DATA_BLOCK "DB_Z220_3_HMI"
{ DB_Accessible_From_OPC_UA := 'FALSE' ;
 DB_Accessible_From_Webserver := 'FALSE' ;
 S7_Optimized_Access := 'FALSE' }
VERSION : 0.1
NON_RETAIN
   STRUCT
      tAlm : Struct   // HMI Alarms
         tE : Struct   // Emergency alarms
            xSpare_0 : Bool;
            xSpare_1 : Bool;
            xSpare_2 : Bool;
            xSpare_3 : Bool;
            xSpare_4 : Bool;
            xSpare_5 : Bool;
            xSpare_6 : Bool;
            xSpare_7 : Bool;
            xSpare_8 : Bool;
            xSpare_9 : Bool;
            xSpare_10 : Bool;
            xSpare_11 : Bool;
            xSpare_12 : Bool;
            xSpare_13 : Bool;
            xSpare_14 : Bool;
            xSpare_15 : Bool;
            xSpare_16 : Bool;
            xSpare_17 : Bool;
            xSpare_18 : Bool;
            xSpare_19 : Bool;
            xSpare_20 : Bool;
            xSpare_21 : Bool;
            xSpare_22 : Bool;
            xSpare_23 : Bool;
            xSpare_24 : Bool;
            xSpare_25 : Bool;
            xSpare_26 { ExternalAccessible := 'False'; ExternalVisible := 'False'; ExternalWritable := 'False'} : Bool;
            xSpare_27 { ExternalAccessible := 'False'; ExternalVisible := 'False'; ExternalWritable := 'False'} : Bool;
            xSpare_28 { ExternalAccessible := 'False'; ExternalVisible := 'False'; ExternalWritable := 'False'} : Bool;
            xSpare_29 { ExternalAccessible := 'False'; ExternalVisible := 'False'; ExternalWritable := 'False'} : Bool;
            xSpare_30 { ExternalAccessible := 'False'; ExternalVisible := 'False'; ExternalWritable := 'False'} : Bool;
            xSpare_31 { ExternalAccessible := 'False'; ExternalVisible := 'False'; ExternalWritable := 'False'} : Bool;
         END_STRUCT;
         tS : Struct   // Stopping faults
            xSpare_0 : Bool;   //
            xSpare_1 : Bool;
            xSpare_2 : Bool;
            xSpare_3 : Bool;
            xSpare_4 : Bool;
            xSpare_5 : Bool;
            xSpare_6 : Bool;
            xSpare_7 : Bool;
            xSpare_8 : Bool;
            xSpare_9 : Bool;
            xSpare_10 : Bool;
            xSpare_11 : Bool;
            xSpare_12 : Bool;
            xSpare_13 : Bool;
            xSpare_14 : Bool;
            xSpare_15 : Bool;
            xSpare_16 : Bool;
            xSpare_17 : Bool;
            xSpare_18 : Bool;
            xSpare_19 : Bool;
            xSpare_20 : Bool;
            xSpare_21 : Bool;
            xSpare_22 : Bool;
            xSpare_23 : Bool;
            xSpare_24 : Bool;
            xSpare_25 : Bool;
            xSpare_26 : Bool;
            xSpare_27 : Bool;
            xSpare_28 : Bool;
            xSpare_29 : Bool;
            xSpare_30 : Bool;
            xSpare_31 : Bool;
         END_STRUCT;
         tF : Struct   // Faults
            x0 : Bool;   // B.Check spray ink carriage
            x2 : Bool;   // SL.Ink tank empty
            x1 : Bool;   // B.Check spray ink carriage dirty lens
            xSpare_3 : Bool;
            xSpare_4 : Bool;
            xSpare_5 : Bool;
            xSpare_6 : Bool;
            xSpare_7 : Bool;
            xSpare_8 : Bool;
            xSpare_9 : Bool;
            xSpare_10 : Bool;
            xSpare_11 : Bool;
            xSpare_12 : Bool;
            xSpare_13 : Bool;
            xSpare_14 : Bool;
            xSpare_15 : Bool;
            xSpare_16 : Bool;
            xSpare_17 : Bool;   //
            xSpare_18 : Bool;
            xSpare_19 : Bool;
            xSpare_20 : Bool;
            xSpare_21 : Bool;
            xSpare_22 : Bool;
            xSpare_23 : Bool;
            xSpare_24 : Bool;
            xSpare_25 : Bool;
            xSpare_26 : Bool;
            xSpare_27 : Bool;
            xSpare_28 : Bool;
            xSpare_29 : Bool;
            xSpare_30 : Bool;
            xSpare_31 : Bool;
         END_STRUCT;
         tW : Struct   // Warnings
            xSpare_0 : Bool;
            xSpare_1 : Bool;
            xSpare_2 : Bool;
            xSpare_3 : Bool;
            xSpare_4 : Bool;
            xSpare_5 : Bool;
            xSpare_6 : Bool;
            xSpare_7 : Bool;
            xSpare_8 : Bool;
            xSpare_9 : Bool;
            xSpare_10 : Bool;
            xSpare_11 : Bool;
            xSpare_12 : Bool;
            xSpare_13 : Bool;
            xSpare_14 : Bool;
            xSpare_15 : Bool;
            xSpare_16 : Bool;
            xSpare_17 : Bool;
            xSpare_18 : Bool;
            xSpare_19 : Bool;
            xSpare_20 : Bool;
            xSpare_21 : Bool;
            xSpare_22 : Bool;
            xSpare_23 : Bool;
            xSpare_24 : Bool;
            xSpare_25 : Bool;
            xSpare_26 : Bool;
            xSpare_27 : Bool;
            xSpare_28 : Bool;
            xSpare_29 : Bool;
            xSpare_30 : Bool;
            xSpare_31 : Bool;
         END_STRUCT;
      END_STRUCT;
      tHMR { ExternalWritable := 'False'} : Struct   // HMI Read
         xSpare0 { ExternalWritable := 'False'} : Bool;
         xSpare1 { ExternalWritable := 'False'} : Bool;
         xSpare2 { ExternalWritable := 'False'} : Bool;
         xSpare3 { ExternalWritable := 'False'} : Bool;
         xSpare4 { ExternalWritable := 'False'} : Bool;
         xSpare5 { ExternalWritable := 'False'} : Bool;
         xSpare6 { ExternalWritable := 'False'} : Bool;
         xSpare7 { ExternalWritable := 'False'} : Bool;
         xSpare8 { ExternalWritable := 'False'} : Bool;
         xSpare9 { ExternalWritable := 'False'} : Bool;
         xSpare10 { ExternalWritable := 'False'} : Bool;
         xSpare11 { ExternalWritable := 'False'} : Bool;
         xSpare12 { ExternalWritable := 'False'} : Bool;
         xSpare13 { ExternalWritable := 'False'} : Bool;
         xSpare14 { ExternalWritable := 'False'} : Bool;
         xSpare15 { ExternalWritable := 'False'} : Bool;   //
         xSpare16 { ExternalWritable := 'False'} : Bool;
         xSpare17 { ExternalWritable := 'False'} : Bool;
         xSpare18 { ExternalWritable := 'False'} : Bool;
         xSpare19 { ExternalWritable := 'False'} : Bool;
         xSpare20 { ExternalWritable := 'False'} : Bool;
         xSpare21 { ExternalWritable := 'False'} : Bool;
         xSpare22 { ExternalWritable := 'False'} : Bool;
         xSpare23 { ExternalWritable := 'False'} : Bool;
         xSpare24 { ExternalWritable := 'False'} : Bool;
         xSpare25 { ExternalWritable := 'False'} : Bool;
         xSpare26 { ExternalWritable := 'False'} : Bool;
         xSpare27 { ExternalWritable := 'False'} : Bool;
         xSpare28 { ExternalWritable := 'False'} : Bool;
         xSpare29 { ExternalWritable := 'False'} : Bool;
         xSpare30 { ExternalWritable := 'False'} : Bool;
         xSpare31 { ExternalWritable := 'False'} : Bool;
         xSpare { ExternalWritable := 'False'} : Array[0..15] of Bool;
         iSpare0 { ExternalWritable := 'False'} : Int;
         iSpare1 { ExternalWritable := 'False'} : Int;
         iSpare2 { ExternalWritable := 'False'} : Int;
         iSpare3 { ExternalWritable := 'False'} : Int;
         iSpare4 { ExternalWritable := 'False'} : Int;
         iSpare5 { ExternalWritable := 'False'} : Int;
         iSpare6 { ExternalWritable := 'False'} : Int;
         iSpare7 { ExternalWritable := 'False'} : Int;
         iSpare8 { ExternalWritable := 'False'} : Int;
         iSpare9 { ExternalWritable := 'False'} : Int;
         iSpare10 { ExternalWritable := 'False'} : Int;
         iSpare11 { ExternalWritable := 'False'} : Int;
         iSpare12 { ExternalWritable := 'False'} : Int;
         iSpare13 { ExternalWritable := 'False'} : Int;
         iSpare14 { ExternalWritable := 'False'} : Int;
         iSpare15 { ExternalWritable := 'False'} : Int;
         iSpare16 { ExternalWritable := 'False'} : Int;
         dZoneMode { ExternalWritable := 'False'} : DInt;   // Zone modality (1=Manual;4=Automatic;8=Manual request) {x|x|x|x|O}
         dProdModeRequest { ExternalWritable := 'False'} : DInt;   // Production modality request (1=Out of Production 3= In production) {x|x|x|x|O}
         dProdModeActual { ExternalWritable := 'False'} : DInt;   // Production modality actual (1=Out of production 3=In production 8=Out of production request 9=In production request) {x|x|x|x|O}
         dActualDistanceFromSnaproll { ExternalWritable := 'False'} : DInt;   // Actual distance from snaproll [mm/100] {x|x|x|x|O}
         dSprayCounter { ExternalWritable := 'False'} : DInt;
         dPhSprayCounter { ExternalWritable := 'False'} : DInt;
         dEvReactionTime { ExternalWritable := 'False'} : DInt;
         dCalibDeltaXPosition_cmm { ExternalWritable := 'False'} : DInt;   // Calibration.Theorical spray position X [mm/100] {mm/100|mm|0|7000|M}
         dCalibDeltaYPosition_cmm { ExternalWritable := 'False'} : DInt;   // Calibration.Theorical spray position Y [mm/100] {mm/100|mm|0|7000|M}
         dSpare9 { ExternalWritable := 'False'} : DInt;
         dSpare10 { ExternalWritable := 'False'} : DInt;
         dSpare11 { ExternalWritable := 'False'} : DInt;
         dSpare12 { ExternalWritable := 'False'} : DInt;
         dSpare13 { ExternalWritable := 'False'} : DInt;
         dSpare14 { ExternalWritable := 'False'} : DInt;
         dSpare15 { ExternalWritable := 'False'} : DInt;
         rSpare0 { ExternalWritable := 'False'} : Real;
         rSpare1 { ExternalWritable := 'False'} : Real;
         rSpare2 { ExternalWritable := 'False'} : Real;
         rSpare3 { ExternalWritable := 'False'} : Real;
         rSpare4 { ExternalWritable := 'False'} : Real;
         rSpare5 { ExternalWritable := 'False'} : Real;
         rSpare6 { ExternalWritable := 'False'} : Real;
         rSpare7 { ExternalWritable := 'False'} : Real;
         rSpare8 { ExternalWritable := 'False'} : Real;
         tManCmd { ExternalWritable := 'False'} : Struct
            xSpare0 { ExternalWritable := 'False'} : Bool;   //
            xSpare1 { ExternalWritable := 'False'} : Bool;
            xSpare2 { ExternalWritable := 'False'} : Bool;
            xSpare3 { ExternalWritable := 'False'} : Bool;
            xSpare4 { ExternalWritable := 'False'} : Bool;
            xSpare5 { ExternalWritable := 'False'} : Bool;
            xSpare6 { ExternalWritable := 'False'} : Bool;
            xSpare7 { ExternalWritable := 'False'} : Bool;
            xSpare8 { ExternalWritable := 'False'} : Bool;
            xSpare9 { ExternalWritable := 'False'} : Bool;
            xSpare10 { ExternalWritable := 'False'} : Bool;
            xSpare11 { ExternalWritable := 'False'} : Bool;
            xSpare12 { ExternalWritable := 'False'} : Bool;
            xSpare13 { ExternalWritable := 'False'} : Bool;
            xSpare14 { ExternalWritable := 'False'} : Bool;
            xSpare15 { ExternalWritable := 'False'} : Bool;
            xSpare { ExternalWritable := 'False'} : Array[0..15] of Bool;
         END_STRUCT;
      END_STRUCT;
      tHMW : Struct   // HMI Write
         xAutoModeReq : Bool;   // Automatic mode request {x|x|x|x|O}
         xManModeReq : Bool;   // Manual mode request {x|x|x|x|O}
         xUpdateDistanceFromSnapRoll : Bool;   // Update Distance From Snap Roll {x|x|x|x|M}
         xCalibrate : Bool;   // Calibrate spray position {x|x|x|x|M}
         xCleaningCycle : Bool;   // Cleaning cycle enabled {x|x|x|x|O}
         xSprayOnBreakEnabled : Bool;   // Spray during glass break {x|x|x|x|O}
         xSprayCheckEnabled : Bool;   // Spray check enabled {x|x|x|x|O}
         xResetCounter : Bool;
         xSpare8 : Bool;
         xSpare9 { ExternalWritable := 'False'} : Bool;
         xSpare10 : Bool;
         xSpare11 : Bool;
         xSpare12 : Bool;
         xSpare13 : Bool;
         xSpare14 : Bool;
         xSpare15 : Bool;   //
         xSpare16 : Bool;   //
         xSpare17 : Bool;
         xSpare18 : Bool;
         xSpare19 : Bool;
         xSpare20 : Bool;
         xSpare21 : Bool;
         xSpare22 : Bool;
         xSpare23 : Bool;
         xSpare24 : Bool;
         xSpare25 : Bool;
         xSpare26 : Bool;
         xSpare27 : Bool;
         xSpare28 : Bool;
         xSpare29 : Bool;
         xSpare30 : Bool;
         xSpare31 : Bool;
         xSpare : Array[0..15] of Bool;
         iSpare0 : Int;
         iSpare1 : Int;
         iSpare2 : Int;
         iSpare3 : Int;
         iSpare4 : Int;
         iSpare5 : Int;
         iSpare6 : Int;
         iSpare7 : Int;
         iSpare8 : Int;
         iSpare9 : Int;
         iSpare10 : Int;
         iSpare11 : Int;
         iSpare12 : Int;
         iSpare13 : Int;
         iSpare14 : Int;
         iSpare15 : Int;
         iSpare16 : Int;
         dDistanceFromSnaproll_cmm : DInt;   // Distance from snaproll [mm/100] {x|x|x|x|O}
         dSpare1 : DInt;   //
         dCleaningInterval_ms : DInt;   // Cleaning cycle interval [ms] {ms|s|3600|36000|O}
         dSpraySpace_cmm : DInt;   // Spray space [mm/100] {mm/100|mm|1|100|O}
         dSprayReactionTimeON_ms : DInt;   // Spray reaction time [ms] {ms|s|0.001|2|M}
         dSprayReactionTimeOFF_ms : DInt;   // Spray reaction time off [ms] {ms|s|0.001|2|M}
         dCalibDefectMeasXPosition_cmm : DInt;   // Calibration.Measured defect position X [mm/100] {mm/100|mm|0|7000|M}
         dCalibSprayMeasXPosition_cmm : DInt;   // Calibration.Measured spray position X [mm/100] {mm/100|mm|0|7000|M}
         dCalibDefectMeasYPosition_cmm : DInt;   // Calibration.Measured defect position Y [mm/100] {mm/100|mm|0|7000|M}
         dCalibSprayMeasYPosition_cmm : DInt;   // Calibration.Measured spray position Y [mm/100] {mm/100|mm|0|7000|M}
         dSpare10 : DInt;
         dSpare11 : DInt;
         dSpare12 : DInt;
         dSpare13 : DInt;
         dSpare14 : DInt;
         dSpare15 : DInt;
         dSpare16 : DInt;
         rSpare0 : Real;
         rSpare1 : Real;
         rSpare2 : Real;
         rSpare3 : Real;
         rSpare4 : Real;
         rSpare5 : Real;
         rSpare6 : Real;
         rSpare7 : Real;
         rSpare8 : Real;
         tManCmd : Struct
            xSpare0 : Bool;
            xSpare1 : Bool;
            xSpare2 { ExternalWritable := 'False'} : Bool;
            xSpare3 { ExternalWritable := 'False'} : Bool;
            xSpare4 { ExternalWritable := 'False'} : Bool;
            xSpare5 { ExternalWritable := 'False'} : Bool;
            xSpare6 { ExternalWritable := 'False'} : Bool;
            xSpare7 { ExternalWritable := 'False'} : Bool;
            xSpare8 { ExternalWritable := 'False'} : Bool;
            xSpare9 { ExternalWritable := 'False'} : Bool;
            xSpare10 { ExternalWritable := 'False'} : Bool;
            xSpare11 { ExternalWritable := 'False'} : Bool;
            xSpare12 { ExternalWritable := 'False'} : Bool;
            xSpare13 { ExternalWritable := 'False'} : Bool;
            xSpare14 { ExternalWritable := 'False'} : Bool;
            xSpare15 { ExternalWritable := 'False'} : Bool;
            xSpare16 : Bool;
            xSpare17 : Bool;
            xSpare18 : Bool;
            xSpare19 : Bool;
            xSpare20 : Bool;
            xSpare21 : Bool;
            xSpare22 : Bool;
            xSpare23 : Bool;
            xSpare24 : Bool;
            xSpare25 : Bool;
            xSpare26 : Bool;
            xSpare27 : Bool;
            xSpare28 : Bool;
            xSpare29 : Bool;
            xSpare30 : Bool;
            xSpare31 : Bool;
         END_STRUCT;
      END_STRUCT;
   END_STRUCT;


BEGIN
   tAlm.tE.xSpare_0 := TRUE;
   tAlm.tE.xSpare_1 := TRUE;
   tAlm.tE.xSpare_2 := TRUE;
   tAlm.tE.xSpare_3 := TRUE;
   tAlm.tE.xSpare_4 := TRUE;
   tAlm.tE.xSpare_5 := TRUE;
   tAlm.tE.xSpare_6 := TRUE;
   tAlm.tE.xSpare_7 := TRUE;
   tAlm.tE.xSpare_8 := TRUE;
   tAlm.tE.xSpare_9 := TRUE;
   tAlm.tE.xSpare_10 := FALSE;
   tAlm.tE.xSpare_11 := FALSE;
   tAlm.tE.xSpare_12 := FALSE;
   tAlm.tE.xSpare_13 := FALSE;
   tAlm.tE.xSpare_14 := FALSE;
   tAlm.tE.xSpare_15 := FALSE;
   tAlm.tE.xSpare_16 := FALSE;
   tAlm.tE.xSpare_17 := FALSE;
   tAlm.tE.xSpare_18 := FALSE;
   tAlm.tE.xSpare_19 := FALSE;
   tAlm.tE.xSpare_20 := FALSE;
   tAlm.tE.xSpare_21 := FALSE;
   tAlm.tE.xSpare_22 := FALSE;
   tAlm.tE.xSpare_23 := FALSE;
   tAlm.tE.xSpare_24 := FALSE;
   tAlm.tE.xSpare_25 := FALSE;
   tAlm.tE.xSpare_26 := FALSE;
   tAlm.tE.xSpare_27 := FALSE;
   tAlm.tE.xSpare_28 := FALSE;
   tAlm.tE.xSpare_29 := FALSE;
   tAlm.tE.xSpare_30 := FALSE;
   tAlm.tE.xSpare_31 := FALSE;
   tAlm.tS.xSpare_0 := FALSE;
   tAlm.tS.xSpare_1 := FALSE;
   tAlm.tS.xSpare_2 := FALSE;
   tAlm.tS.xSpare_3 := FALSE;
   tAlm.tS.xSpare_4 := FALSE;
   tAlm.tS.xSpare_5 := FALSE;
   tAlm.tS.xSpare_6 := FALSE;
   tAlm.tS.xSpare_7 := FALSE;
   tAlm.tS.xSpare_8 := FALSE;
   tAlm.tS.xSpare_9 := FALSE;
   tAlm.tS.xSpare_10 := FALSE;
   tAlm.tS.xSpare_11 := FALSE;
   tAlm.tS.xSpare_12 := FALSE;
   tAlm.tS.xSpare_13 := FALSE;
   tAlm.tS.xSpare_14 := FALSE;
   tAlm.tS.xSpare_15 := FALSE;
   tAlm.tS.xSpare_16 := FALSE;
   tAlm.tS.xSpare_17 := FALSE;
   tAlm.tS.xSpare_18 := FALSE;
   tAlm.tS.xSpare_19 := FALSE;
   tAlm.tS.xSpare_20 := FALSE;
   tAlm.tS.xSpare_21 := FALSE;
   tAlm.tS.xSpare_22 := FALSE;
   tAlm.tS.xSpare_23 := FALSE;
   tAlm.tS.xSpare_24 := FALSE;
   tAlm.tS.xSpare_25 := FALSE;
   tAlm.tS.xSpare_26 := FALSE;
   tAlm.tS.xSpare_27 := FALSE;
   tAlm.tS.xSpare_28 := FALSE;
   tAlm.tS.xSpare_29 := FALSE;
   tAlm.tS.xSpare_30 := FALSE;
   tAlm.tS.xSpare_31 := FALSE;
   tAlm.tF.xSpare_3 := FALSE;
   tAlm.tF.xSpare_4 := FALSE;
   tAlm.tF.xSpare_5 := FALSE;
   tAlm.tF.xSpare_6 := FALSE;
   tAlm.tF.xSpare_7 := FALSE;
   tAlm.tF.xSpare_8 := FALSE;
   tAlm.tF.xSpare_9 := FALSE;
   tAlm.tF.xSpare_10 := FALSE;
   tAlm.tF.xSpare_11 := FALSE;
   tAlm.tF.xSpare_20 := FALSE;
   tAlm.tF.xSpare_21 := FALSE;
   tAlm.tF.xSpare_22 := FALSE;
   tAlm.tF.xSpare_23 := FALSE;
   tAlm.tF.xSpare_24 := FALSE;
   tAlm.tF.xSpare_25 := FALSE;
   tAlm.tF.xSpare_26 := FALSE;
   tAlm.tF.xSpare_27 := FALSE;
   tAlm.tF.xSpare_28 := FALSE;
   tAlm.tF.xSpare_29 := FALSE;
   tAlm.tF.xSpare_30 := FALSE;
   tAlm.tF.xSpare_31 := FALSE;
   tAlm.tW.xSpare_0 := FALSE;
   tAlm.tW.xSpare_1 := FALSE;
   tAlm.tW.xSpare_2 := FALSE;
   tAlm.tW.xSpare_3 := FALSE;
   tAlm.tW.xSpare_4 := FALSE;
   tAlm.tW.xSpare_5 := FALSE;
   tAlm.tW.xSpare_6 := FALSE;
   tAlm.tW.xSpare_7 := FALSE;
   tAlm.tW.xSpare_8 := FALSE;
   tAlm.tW.xSpare_9 := FALSE;
   tAlm.tW.xSpare_10 := FALSE;
   tAlm.tW.xSpare_11 := FALSE;
   tAlm.tW.xSpare_12 := FALSE;
   tAlm.tW.xSpare_13 := FALSE;
   tAlm.tW.xSpare_14 := FALSE;
   tAlm.tW.xSpare_15 := FALSE;
   tAlm.tW.xSpare_16 := FALSE;
   tAlm.tW.xSpare_17 := FALSE;
   tAlm.tW.xSpare_18 := FALSE;
   tAlm.tW.xSpare_19 := FALSE;
   tAlm.tW.xSpare_20 := FALSE;
   tAlm.tW.xSpare_21 := FALSE;
   tAlm.tW.xSpare_22 := FALSE;
   tAlm.tW.xSpare_23 := FALSE;
   tAlm.tW.xSpare_24 := FALSE;
   tAlm.tW.xSpare_25 := FALSE;
   tAlm.tW.xSpare_26 := FALSE;
   tAlm.tW.xSpare_27 := FALSE;
   tAlm.tW.xSpare_28 := FALSE;
   tAlm.tW.xSpare_29 := FALSE;
   tAlm.tW.xSpare_30 := FALSE;
   tAlm.tW.xSpare_31 := FALSE;
   tHMR.xSpare15 := FALSE;
   tHMW.xSpare15 := FALSE;
   tHMW.xSpare16 := FALSE;

END_DATA_BLOCK

DATA_BLOCK "DB_Z220_2_HMI"
{ DB_Accessible_From_OPC_UA := 'FALSE' ;
 DB_Accessible_From_Webserver := 'FALSE' ;
 S7_Optimized_Access := 'FALSE' }
VERSION : 0.1
NON_RETAIN
   STRUCT
      tAlm : Struct   // HMI Alarms
         tE : Struct   // Emergency alarms
            xSpare_0 : Bool;
            xSpare_1 : Bool;
            xSpare_2 : Bool;
            xSpare_3 : Bool;
            xSpare_4 : Bool;
            xSpare_5 : Bool;
            xSpare_6 : Bool;
            xSpare_7 : Bool;
            xSpare_8 : Bool;
            xSpare_9 : Bool;
            xSpare_10 : Bool;
            xSpare_11 : Bool;
            xSpare_12 : Bool;
            xSpare_13 : Bool;
            xSpare_14 : Bool;
            xSpare_15 : Bool;
            xSpare_16 : Bool;
            xSpare_17 : Bool;
            xSpare_18 : Bool;
            xSpare_19 : Bool;
            xSpare_20 : Bool;
            xSpare_21 : Bool;
            xSpare_22 : Bool;
            xSpare_23 : Bool;
            xSpare_24 : Bool;
            xSpare_25 : Bool;
            xSpare_26 { ExternalAccessible := 'False'; ExternalVisible := 'False'; ExternalWritable := 'False'} : Bool;
            xSpare_27 { ExternalAccessible := 'False'; ExternalVisible := 'False'; ExternalWritable := 'False'} : Bool;
            xSpare_28 { ExternalAccessible := 'False'; ExternalVisible := 'False'; ExternalWritable := 'False'} : Bool;
            xSpare_29 { ExternalAccessible := 'False'; ExternalVisible := 'False'; ExternalWritable := 'False'} : Bool;
            xSpare_30 { ExternalAccessible := 'False'; ExternalVisible := 'False'; ExternalWritable := 'False'} : Bool;
            xSpare_31 { ExternalAccessible := 'False'; ExternalVisible := 'False'; ExternalWritable := 'False'} : Bool;
         END_STRUCT;
         tS : Struct   // Stopping faults
            xSpare_0 : Bool;   //
            xSpare_1 : Bool;
            xSpare_2 : Bool;
            xSpare_3 : Bool;
            xSpare_4 : Bool;
            xSpare_5 : Bool;
            xSpare_6 : Bool;
            xSpare_7 : Bool;
            xSpare_8 : Bool;
            xSpare_9 : Bool;
            xSpare_10 : Bool;
            xSpare_11 : Bool;
            xSpare_12 : Bool;
            xSpare_13 : Bool;
            xSpare_14 : Bool;
            xSpare_15 : Bool;
            xSpare_16 : Bool;
            xSpare_17 : Bool;
            xSpare_18 : Bool;
            xSpare_19 : Bool;
            xSpare_20 : Bool;
            xSpare_21 : Bool;
            xSpare_22 : Bool;
            xSpare_23 : Bool;
            xSpare_24 : Bool;
            xSpare_25 : Bool;
            xSpare_26 : Bool;
            xSpare_27 : Bool;
            xSpare_28 : Bool;
            xSpare_29 : Bool;
            xSpare_30 : Bool;
            xSpare_31 : Bool;
         END_STRUCT;
         tF : Struct   // Faults
            x0 : Bool;   // B.Check spray ink carriage
            x2 : Bool;   // SL.Ink tank empty
            x1 : Bool;   // B.Check spray ink carriage dirty lens
            xSpare_3 : Bool;
            xSpare_4 : Bool;
            xSpare_5 : Bool;
            xSpare_6 : Bool;
            xSpare_7 : Bool;
            xSpare_8 : Bool;
            xSpare_9 : Bool;
            xSpare_10 : Bool;
            xSpare_11 : Bool;
            xSpare_12 : Bool;
            xSpare_13 : Bool;
            xSpare_14 : Bool;
            xSpare_15 : Bool;
            xSpare_16 : Bool;
            xSpare_17 : Bool;   //
            xSpare_18 : Bool;
            xSpare_19 : Bool;
            xSpare_20 : Bool;
            xSpare_21 : Bool;
            xSpare_22 : Bool;
            xSpare_23 : Bool;
            xSpare_24 : Bool;
            xSpare_25 : Bool;
            xSpare_26 : Bool;
            xSpare_27 : Bool;
            xSpare_28 : Bool;
            xSpare_29 : Bool;
            xSpare_30 : Bool;
            xSpare_31 : Bool;
         END_STRUCT;
         tW : Struct   // Warnings
            xSpare_0 : Bool;
            xSpare_1 : Bool;
            xSpare_2 : Bool;
            xSpare_3 : Bool;
            xSpare_4 : Bool;
            xSpare_5 : Bool;
            xSpare_6 : Bool;
            xSpare_7 : Bool;
            xSpare_8 : Bool;
            xSpare_9 : Bool;
            xSpare_10 : Bool;
            xSpare_11 : Bool;
            xSpare_12 : Bool;
            xSpare_13 : Bool;
            xSpare_14 : Bool;
            xSpare_15 : Bool;
            xSpare_16 : Bool;
            xSpare_17 : Bool;
            xSpare_18 : Bool;
            xSpare_19 : Bool;
            xSpare_20 : Bool;
            xSpare_21 : Bool;
            xSpare_22 : Bool;
            xSpare_23 : Bool;
            xSpare_24 : Bool;
            xSpare_25 : Bool;
            xSpare_26 : Bool;
            xSpare_27 : Bool;
            xSpare_28 : Bool;
            xSpare_29 : Bool;
            xSpare_30 : Bool;
            xSpare_31 : Bool;
         END_STRUCT;
      END_STRUCT;
      tHMR { ExternalWritable := 'False'} : Struct   // HMI Read
         xSpare0 { ExternalWritable := 'False'} : Bool;
         xSpare1 { ExternalWritable := 'False'} : Bool;
         xSpare2 { ExternalWritable := 'False'} : Bool;
         xSpare3 { ExternalWritable := 'False'} : Bool;
         xSpare4 { ExternalWritable := 'False'} : Bool;
         xSpare5 { ExternalWritable := 'False'} : Bool;
         xSpare6 { ExternalWritable := 'False'} : Bool;
         xSpare7 { ExternalWritable := 'False'} : Bool;
         xSpare8 { ExternalWritable := 'False'} : Bool;
         xSpare9 { ExternalWritable := 'False'} : Bool;
         xSpare10 { ExternalWritable := 'False'} : Bool;
         xSpare11 { ExternalWritable := 'False'} : Bool;
         xSpare12 { ExternalWritable := 'False'} : Bool;
         xSpare13 { ExternalWritable := 'False'} : Bool;
         xSpare14 { ExternalWritable := 'False'} : Bool;
         xSpare15 { ExternalWritable := 'False'} : Bool;   //
         xSpare16 { ExternalWritable := 'False'} : Bool;
         xSpare17 { ExternalWritable := 'False'} : Bool;
         xSpare18 { ExternalWritable := 'False'} : Bool;
         xSpare19 { ExternalWritable := 'False'} : Bool;
         xSpare20 { ExternalWritable := 'False'} : Bool;
         xSpare21 { ExternalWritable := 'False'} : Bool;
         xSpare22 { ExternalWritable := 'False'} : Bool;
         xSpare23 { ExternalWritable := 'False'} : Bool;
         xSpare24 { ExternalWritable := 'False'} : Bool;
         xSpare25 { ExternalWritable := 'False'} : Bool;
         xSpare26 { ExternalWritable := 'False'} : Bool;
         xSpare27 { ExternalWritable := 'False'} : Bool;
         xSpare28 { ExternalWritable := 'False'} : Bool;
         xSpare29 { ExternalWritable := 'False'} : Bool;
         xSpare30 { ExternalWritable := 'False'} : Bool;
         xSpare31 { ExternalWritable := 'False'} : Bool;
         xSpare { ExternalWritable := 'False'} : Array[0..15] of Bool;
         iSpare0 { ExternalWritable := 'False'} : Int;
         iSpare1 { ExternalWritable := 'False'} : Int;
         iSpare2 { ExternalWritable := 'False'} : Int;
         iSpare3 { ExternalWritable := 'False'} : Int;
         iSpare4 { ExternalWritable := 'False'} : Int;
         iSpare5 { ExternalWritable := 'False'} : Int;
         iSpare6 { ExternalWritable := 'False'} : Int;
         iSpare7 { ExternalWritable := 'False'} : Int;
         iSpare8 { ExternalWritable := 'False'} : Int;
         iSpare9 { ExternalWritable := 'False'} : Int;
         iSpare10 { ExternalWritable := 'False'} : Int;
         iSpare11 { ExternalWritable := 'False'} : Int;
         iSpare12 { ExternalWritable := 'False'} : Int;
         iSpare13 { ExternalWritable := 'False'} : Int;
         iSpare14 { ExternalWritable := 'False'} : Int;
         iSpare15 { ExternalWritable := 'False'} : Int;
         iSpare16 { ExternalWritable := 'False'} : Int;
         dZoneMode { ExternalWritable := 'False'} : DInt;   // Zone modality (1=Manual;4=Automatic;8=Manual request) {x|x|x|x|O}
         dProdModeRequest { ExternalWritable := 'False'} : DInt;   // Production modality request (1=Out of Production 3= In production) {x|x|x|x|O}
         dProdModeActual { ExternalWritable := 'False'} : DInt;   // Production modality actual (1=Out of production 3=In production 8=Out of production request 9=In production request) {x|x|x|x|O}
         dActualDistanceFromSnaproll { ExternalWritable := 'False'} : DInt;   // Actual distance from snaproll [mm/100] {x|x|x|x|O}
         dSprayCounter { ExternalWritable := 'False'} : DInt;
         dPhSprayCounter { ExternalWritable := 'False'} : DInt;
         dEvReactionTime { ExternalWritable := 'False'} : DInt;
         dCalibDeltaXPosition_cmm { ExternalWritable := 'False'} : DInt;   // Calibration.Theorical spray position X [mm/100] {mm/100|mm|0|7000|M}
         dCalibDeltaYPosition_cmm { ExternalWritable := 'False'} : DInt;   // Calibration.Theorical spray position Y [mm/100] {mm/100|mm|0|7000|M}
         dSpare9 { ExternalWritable := 'False'} : DInt;
         dSpare10 { ExternalWritable := 'False'} : DInt;
         dSpare11 { ExternalWritable := 'False'} : DInt;
         dSpare12 { ExternalWritable := 'False'} : DInt;
         dSpare13 { ExternalWritable := 'False'} : DInt;
         dSpare14 { ExternalWritable := 'False'} : DInt;
         dSpare15 { ExternalWritable := 'False'} : DInt;
         rSpare0 { ExternalWritable := 'False'} : Real;
         rSpare1 { ExternalWritable := 'False'} : Real;
         rSpare2 { ExternalWritable := 'False'} : Real;
         rSpare3 { ExternalWritable := 'False'} : Real;
         rSpare4 { ExternalWritable := 'False'} : Real;
         rSpare5 { ExternalWritable := 'False'} : Real;
         rSpare6 { ExternalWritable := 'False'} : Real;
         rSpare7 { ExternalWritable := 'False'} : Real;
         rSpare8 { ExternalWritable := 'False'} : Real;
         tManCmd { ExternalWritable := 'False'} : Struct
            xSpare0 { ExternalWritable := 'False'} : Bool;   //
            xSpare1 { ExternalWritable := 'False'} : Bool;
            xSpare2 { ExternalWritable := 'False'} : Bool;
            xSpare3 { ExternalWritable := 'False'} : Bool;
            xSpare4 { ExternalWritable := 'False'} : Bool;
            xSpare5 { ExternalWritable := 'False'} : Bool;
            xSpare6 { ExternalWritable := 'False'} : Bool;
            xSpare7 { ExternalWritable := 'False'} : Bool;
            xSpare8 { ExternalWritable := 'False'} : Bool;
            xSpare9 { ExternalWritable := 'False'} : Bool;
            xSpare10 { ExternalWritable := 'False'} : Bool;
            xSpare11 { ExternalWritable := 'False'} : Bool;
            xSpare12 { ExternalWritable := 'False'} : Bool;
            xSpare13 { ExternalWritable := 'False'} : Bool;
            xSpare14 { ExternalWritable := 'False'} : Bool;
            xSpare15 { ExternalWritable := 'False'} : Bool;
            xSpare { ExternalWritable := 'False'} : Array[0..15] of Bool;
         END_STRUCT;
      END_STRUCT;
      tHMW : Struct   // HMI Write
         xAutoModeReq : Bool;   // Automatic mode request {x|x|x|x|O}
         xManModeReq : Bool;   // Manual mode request {x|x|x|x|O}
         xUpdateDistanceFromSnapRoll : Bool;   // Update Distance From Snap Roll {x|x|x|x|M}
         xCalibrate : Bool;   // Calibrate spray position {x|x|x|x|M}
         xCleaningCycle : Bool;   // Cleaning cycle enabled {x|x|x|x|O}
         xSprayOnBreakEnabled : Bool;   // Spray during glass break {x|x|x|x|O}
         xSprayCheckEnabled : Bool;   // Spray check enabled {x|x|x|x|O}
         xResetCounter : Bool;
         xSpare8 : Bool;
         xSpare9 { ExternalWritable := 'False'} : Bool;
         xSpare10 : Bool;
         xSpare11 : Bool;
         xSpare12 : Bool;
         xSpare13 : Bool;
         xSpare14 : Bool;
         xSpare15 : Bool;   //
         xSpare16 : Bool;   //
         xSpare17 : Bool;
         xSpare18 : Bool;
         xSpare19 : Bool;
         xSpare20 : Bool;
         xSpare21 : Bool;
         xSpare22 : Bool;
         xSpare23 : Bool;
         xSpare24 : Bool;
         xSpare25 : Bool;
         xSpare26 : Bool;
         xSpare27 : Bool;
         xSpare28 : Bool;
         xSpare29 : Bool;
         xSpare30 : Bool;
         xSpare31 : Bool;
         xSpare : Array[0..15] of Bool;
         iSpare0 : Int;
         iSpare1 : Int;
         iSpare2 : Int;
         iSpare3 : Int;
         iSpare4 : Int;
         iSpare5 : Int;
         iSpare6 : Int;
         iSpare7 : Int;
         iSpare8 : Int;
         iSpare9 : Int;
         iSpare10 : Int;
         iSpare11 : Int;
         iSpare12 : Int;
         iSpare13 : Int;
         iSpare14 : Int;
         iSpare15 : Int;
         iSpare16 : Int;
         dDistanceFromSnaproll_cmm : DInt;   // Distance from snaproll [mm/100] {x|x|x|x|O}
         dSpare1 : DInt;   //
         dCleaningInterval_ms : DInt;   // Cleaning cycle interval [ms] {ms|s|3600|36000|O}
         dSpraySpace_cmm : DInt;   // Spray space [mm/100] {mm/100|mm|1|100|O}
         dSprayReactionTimeON_ms : DInt;   // Spray reaction time [ms] {ms|s|0.001|2|M}
         dSprayReactionTimeOFF_ms : DInt;   // Spray reaction time off [ms] {ms|s|0.001|2|M}
         dCalibDefectMeasXPosition_cmm : DInt;   // Calibration.Measured defect position X [mm/100] {mm/100|mm|0|7000|M}
         dCalibSprayMeasXPosition_cmm : DInt;   // Calibration.Measured spray position X [mm/100] {mm/100|mm|0|7000|M}
         dCalibDefectMeasYPosition_cmm : DInt;   // Calibration.Measured defect position Y [mm/100] {mm/100|mm|0|7000|M}
         dCalibSprayMeasYPosition_cmm : DInt;   // Calibration.Measured spray position Y [mm/100] {mm/100|mm|0|7000|M}
         dSpare10 : DInt;
         dSpare11 : DInt;
         dSpare12 : DInt;
         dSpare13 : DInt;
         dSpare14 : DInt;
         dSpare15 : DInt;
         dSpare16 : DInt;
         rSpare0 : Real;
         rSpare1 : Real;
         rSpare2 : Real;
         rSpare3 : Real;
         rSpare4 : Real;
         rSpare5 : Real;
         rSpare6 : Real;
         rSpare7 : Real;
         rSpare8 : Real;
         tManCmd : Struct
            xSpare0 : Bool;
            xSpare1 : Bool;
            xSpare2 { ExternalWritable := 'False'} : Bool;
            xSpare3 { ExternalWritable := 'False'} : Bool;
            xSpare4 { ExternalWritable := 'False'} : Bool;
            xSpare5 { ExternalWritable := 'False'} : Bool;
            xSpare6 { ExternalWritable := 'False'} : Bool;
            xSpare7 { ExternalWritable := 'False'} : Bool;
            xSpare8 { ExternalWritable := 'False'} : Bool;
            xSpare9 { ExternalWritable := 'False'} : Bool;
            xSpare10 { ExternalWritable := 'False'} : Bool;
            xSpare11 { ExternalWritable := 'False'} : Bool;
            xSpare12 { ExternalWritable := 'False'} : Bool;
            xSpare13 { ExternalWritable := 'False'} : Bool;
            xSpare14 { ExternalWritable := 'False'} : Bool;
            xSpare15 { ExternalWritable := 'False'} : Bool;
            xSpare16 : Bool;
            xSpare17 : Bool;
            xSpare18 : Bool;
            xSpare19 : Bool;
            xSpare20 : Bool;
            xSpare21 : Bool;
            xSpare22 : Bool;
            xSpare23 : Bool;
            xSpare24 : Bool;
            xSpare25 : Bool;
            xSpare26 : Bool;
            xSpare27 : Bool;
            xSpare28 : Bool;
            xSpare29 : Bool;
            xSpare30 : Bool;
            xSpare31 : Bool;
         END_STRUCT;
      END_STRUCT;
   END_STRUCT;


BEGIN
   tAlm.tE.xSpare_0 := TRUE;
   tAlm.tE.xSpare_1 := TRUE;
   tAlm.tE.xSpare_2 := TRUE;
   tAlm.tE.xSpare_3 := TRUE;
   tAlm.tE.xSpare_4 := TRUE;
   tAlm.tE.xSpare_5 := TRUE;
   tAlm.tE.xSpare_6 := TRUE;
   tAlm.tE.xSpare_7 := TRUE;
   tAlm.tE.xSpare_8 := TRUE;
   tAlm.tE.xSpare_9 := TRUE;
   tAlm.tE.xSpare_10 := FALSE;
   tAlm.tE.xSpare_11 := FALSE;
   tAlm.tE.xSpare_12 := FALSE;
   tAlm.tE.xSpare_13 := FALSE;
   tAlm.tE.xSpare_14 := FALSE;
   tAlm.tE.xSpare_15 := FALSE;
   tAlm.tE.xSpare_16 := FALSE;
   tAlm.tE.xSpare_17 := FALSE;
   tAlm.tE.xSpare_18 := FALSE;
   tAlm.tE.xSpare_19 := FALSE;
   tAlm.tE.xSpare_20 := FALSE;
   tAlm.tE.xSpare_21 := FALSE;
   tAlm.tE.xSpare_22 := FALSE;
   tAlm.tE.xSpare_23 := FALSE;
   tAlm.tE.xSpare_24 := FALSE;
   tAlm.tE.xSpare_25 := FALSE;
   tAlm.tE.xSpare_26 := FALSE;
   tAlm.tE.xSpare_27 := FALSE;
   tAlm.tE.xSpare_28 := FALSE;
   tAlm.tE.xSpare_29 := FALSE;
   tAlm.tE.xSpare_30 := FALSE;
   tAlm.tE.xSpare_31 := FALSE;
   tAlm.tS.xSpare_0 := FALSE;
   tAlm.tS.xSpare_1 := FALSE;
   tAlm.tS.xSpare_2 := FALSE;
   tAlm.tS.xSpare_3 := FALSE;
   tAlm.tS.xSpare_4 := FALSE;
   tAlm.tS.xSpare_5 := FALSE;
   tAlm.tS.xSpare_6 := FALSE;
   tAlm.tS.xSpare_7 := FALSE;
   tAlm.tS.xSpare_8 := FALSE;
   tAlm.tS.xSpare_9 := FALSE;
   tAlm.tS.xSpare_10 := FALSE;
   tAlm.tS.xSpare_11 := FALSE;
   tAlm.tS.xSpare_12 := FALSE;
   tAlm.tS.xSpare_13 := FALSE;
   tAlm.tS.xSpare_14 := FALSE;
   tAlm.tS.xSpare_15 := FALSE;
   tAlm.tS.xSpare_16 := FALSE;
   tAlm.tS.xSpare_17 := FALSE;
   tAlm.tS.xSpare_18 := FALSE;
   tAlm.tS.xSpare_19 := FALSE;
   tAlm.tS.xSpare_20 := FALSE;
   tAlm.tS.xSpare_21 := FALSE;
   tAlm.tS.xSpare_22 := FALSE;
   tAlm.tS.xSpare_23 := FALSE;
   tAlm.tS.xSpare_24 := FALSE;
   tAlm.tS.xSpare_25 := FALSE;
   tAlm.tS.xSpare_26 := FALSE;
   tAlm.tS.xSpare_27 := FALSE;
   tAlm.tS.xSpare_28 := FALSE;
   tAlm.tS.xSpare_29 := FALSE;
   tAlm.tS.xSpare_30 := FALSE;
   tAlm.tS.xSpare_31 := FALSE;
   tAlm.tF.xSpare_3 := FALSE;
   tAlm.tF.xSpare_4 := FALSE;
   tAlm.tF.xSpare_5 := FALSE;
   tAlm.tF.xSpare_6 := FALSE;
   tAlm.tF.xSpare_7 := FALSE;
   tAlm.tF.xSpare_8 := FALSE;
   tAlm.tF.xSpare_9 := FALSE;
   tAlm.tF.xSpare_10 := FALSE;
   tAlm.tF.xSpare_11 := FALSE;
   tAlm.tF.xSpare_20 := FALSE;
   tAlm.tF.xSpare_21 := FALSE;
   tAlm.tF.xSpare_22 := FALSE;
   tAlm.tF.xSpare_23 := FALSE;
   tAlm.tF.xSpare_24 := FALSE;
   tAlm.tF.xSpare_25 := FALSE;
   tAlm.tF.xSpare_26 := FALSE;
   tAlm.tF.xSpare_27 := FALSE;
   tAlm.tF.xSpare_28 := FALSE;
   tAlm.tF.xSpare_29 := FALSE;
   tAlm.tF.xSpare_30 := FALSE;
   tAlm.tF.xSpare_31 := FALSE;
   tAlm.tW.xSpare_0 := FALSE;
   tAlm.tW.xSpare_1 := FALSE;
   tAlm.tW.xSpare_2 := FALSE;
   tAlm.tW.xSpare_3 := FALSE;
   tAlm.tW.xSpare_4 := FALSE;
   tAlm.tW.xSpare_5 := FALSE;
   tAlm.tW.xSpare_6 := FALSE;
   tAlm.tW.xSpare_7 := FALSE;
   tAlm.tW.xSpare_8 := FALSE;
   tAlm.tW.xSpare_9 := FALSE;
   tAlm.tW.xSpare_10 := FALSE;
   tAlm.tW.xSpare_11 := FALSE;
   tAlm.tW.xSpare_12 := FALSE;
   tAlm.tW.xSpare_13 := FALSE;
   tAlm.tW.xSpare_14 := FALSE;
   tAlm.tW.xSpare_15 := FALSE;
   tAlm.tW.xSpare_16 := FALSE;
   tAlm.tW.xSpare_17 := FALSE;
   tAlm.tW.xSpare_18 := FALSE;
   tAlm.tW.xSpare_19 := FALSE;
   tAlm.tW.xSpare_20 := FALSE;
   tAlm.tW.xSpare_21 := FALSE;
   tAlm.tW.xSpare_22 := FALSE;
   tAlm.tW.xSpare_23 := FALSE;
   tAlm.tW.xSpare_24 := FALSE;
   tAlm.tW.xSpare_25 := FALSE;
   tAlm.tW.xSpare_26 := FALSE;
   tAlm.tW.xSpare_27 := FALSE;
   tAlm.tW.xSpare_28 := FALSE;
   tAlm.tW.xSpare_29 := FALSE;
   tAlm.tW.xSpare_30 := FALSE;
   tAlm.tW.xSpare_31 := FALSE;
   tHMR.xSpare15 := FALSE;
   tHMW.xSpare15 := FALSE;
   tHMW.xSpare16 := FALSE;

END_DATA_BLOCK

DATA_BLOCK "DB_Z220_1_HMI"
{ DB_Accessible_From_OPC_UA := 'FALSE' ;
 DB_Accessible_From_Webserver := 'FALSE' ;
 S7_Optimized_Access := 'FALSE' }
VERSION : 0.1
NON_RETAIN
   STRUCT
      tAlm : Struct   // HMI Alarms
         tE : Struct   // Emergency alarms
            xSpare_0 : Bool;
            xSpare_1 : Bool;
            xSpare_2 : Bool;
            xSpare_3 : Bool;
            xSpare_4 : Bool;
            xSpare_5 : Bool;
            xSpare_6 : Bool;
            xSpare_7 : Bool;
            xSpare_8 : Bool;
            xSpare_9 : Bool;
            xSpare_10 : Bool;
            xSpare_11 : Bool;
            xSpare_12 : Bool;
            xSpare_13 : Bool;
            xSpare_14 : Bool;
            xSpare_15 : Bool;
            xSpare_16 : Bool;
            xSpare_17 : Bool;
            xSpare_18 : Bool;
            xSpare_19 : Bool;
            xSpare_20 : Bool;
            xSpare_21 : Bool;
            xSpare_22 : Bool;
            xSpare_23 : Bool;
            xSpare_24 : Bool;
            xSpare_25 : Bool;
            xSpare_26 { ExternalAccessible := 'False'; ExternalVisible := 'False'; ExternalWritable := 'False'} : Bool;
            xSpare_27 { ExternalAccessible := 'False'; ExternalVisible := 'False'; ExternalWritable := 'False'} : Bool;
            xSpare_28 { ExternalAccessible := 'False'; ExternalVisible := 'False'; ExternalWritable := 'False'} : Bool;
            xSpare_29 { ExternalAccessible := 'False'; ExternalVisible := 'False'; ExternalWritable := 'False'} : Bool;
            xSpare_30 { ExternalAccessible := 'False'; ExternalVisible := 'False'; ExternalWritable := 'False'} : Bool;
            xSpare_31 { ExternalAccessible := 'False'; ExternalVisible := 'False'; ExternalWritable := 'False'} : Bool;
         END_STRUCT;
         tS : Struct   // Stopping faults
            xSpare_0 : Bool;   //
            xSpare_1 : Bool;
            xSpare_2 : Bool;
            xSpare_3 : Bool;
            xSpare_4 : Bool;
            xSpare_5 : Bool;
            xSpare_6 : Bool;
            xSpare_7 : Bool;
            xSpare_8 : Bool;
            xSpare_9 : Bool;
            xSpare_10 : Bool;
            xSpare_11 : Bool;
            xSpare_12 : Bool;
            xSpare_13 : Bool;
            xSpare_14 : Bool;
            xSpare_15 : Bool;
            xSpare_16 : Bool;
            xSpare_17 : Bool;
            xSpare_18 : Bool;
            xSpare_19 : Bool;
            xSpare_20 : Bool;
            xSpare_21 : Bool;
            xSpare_22 : Bool;
            xSpare_23 : Bool;
            xSpare_24 : Bool;
            xSpare_25 : Bool;
            xSpare_26 : Bool;
            xSpare_27 : Bool;
            xSpare_28 : Bool;
            xSpare_29 : Bool;
            xSpare_30 : Bool;
            xSpare_31 : Bool;
         END_STRUCT;
         tF : Struct   // Faults
            x0 : Bool;   // B.Check spray ink carriage
            x2 : Bool;   // SL.Ink tank empty
            x1 : Bool;   // B.Check spray ink carriage dirty lens
            xSpare_3 : Bool;
            xSpare_4 : Bool;
            xSpare_5 : Bool;
            xSpare_6 : Bool;
            xSpare_7 : Bool;
            xSpare_8 : Bool;
            xSpare_9 : Bool;
            xSpare_10 : Bool;
            xSpare_11 : Bool;
            xSpare_12 : Bool;
            xSpare_13 : Bool;
            xSpare_14 : Bool;
            xSpare_15 : Bool;
            xSpare_16 : Bool;
            xSpare_17 : Bool;   //
            xSpare_18 : Bool;
            xSpare_19 : Bool;
            xSpare_20 : Bool;
            xSpare_21 : Bool;
            xSpare_22 : Bool;
            xSpare_23 : Bool;
            xSpare_24 : Bool;
            xSpare_25 : Bool;
            xSpare_26 : Bool;
            xSpare_27 : Bool;
            xSpare_28 : Bool;
            xSpare_29 : Bool;
            xSpare_30 : Bool;
            xSpare_31 : Bool;
         END_STRUCT;
         tW : Struct   // Warnings
            xSpare_0 : Bool;
            xSpare_1 : Bool;
            xSpare_2 : Bool;
            xSpare_3 : Bool;
            xSpare_4 : Bool;
            xSpare_5 : Bool;
            xSpare_6 : Bool;
            xSpare_7 : Bool;
            xSpare_8 : Bool;
            xSpare_9 : Bool;
            xSpare_10 : Bool;
            xSpare_11 : Bool;
            xSpare_12 : Bool;
            xSpare_13 : Bool;
            xSpare_14 : Bool;
            xSpare_15 : Bool;
            xSpare_16 : Bool;
            xSpare_17 : Bool;
            xSpare_18 : Bool;
            xSpare_19 : Bool;
            xSpare_20 : Bool;
            xSpare_21 : Bool;
            xSpare_22 : Bool;
            xSpare_23 : Bool;
            xSpare_24 : Bool;
            xSpare_25 : Bool;
            xSpare_26 : Bool;
            xSpare_27 : Bool;
            xSpare_28 : Bool;
            xSpare_29 : Bool;
            xSpare_30 : Bool;
            xSpare_31 : Bool;
         END_STRUCT;
      END_STRUCT;
      tHMR { ExternalWritable := 'False'} : Struct   // HMI Read
         xSpare0 { ExternalWritable := 'False'} : Bool;
         xSpare1 { ExternalWritable := 'False'} : Bool;
         xSpare2 { ExternalWritable := 'False'} : Bool;
         xSpare3 { ExternalWritable := 'False'} : Bool;
         xSpare4 { ExternalWritable := 'False'} : Bool;
         xSpare5 { ExternalWritable := 'False'} : Bool;
         xSpare6 { ExternalWritable := 'False'} : Bool;
         xSpare7 { ExternalWritable := 'False'} : Bool;
         xSpare8 { ExternalWritable := 'False'} : Bool;
         xSpare9 { ExternalWritable := 'False'} : Bool;
         xSpare10 { ExternalWritable := 'False'} : Bool;
         xSpare11 { ExternalWritable := 'False'} : Bool;
         xSpare12 { ExternalWritable := 'False'} : Bool;
         xSpare13 { ExternalWritable := 'False'} : Bool;
         xSpare14 { ExternalWritable := 'False'} : Bool;
         xSpare15 { ExternalWritable := 'False'} : Bool;   //
         xSpare16 { ExternalWritable := 'False'} : Bool;
         xSpare17 { ExternalWritable := 'False'} : Bool;
         xSpare18 { ExternalWritable := 'False'} : Bool;
         xSpare19 { ExternalWritable := 'False'} : Bool;
         xSpare20 { ExternalWritable := 'False'} : Bool;
         xSpare21 { ExternalWritable := 'False'} : Bool;
         xSpare22 { ExternalWritable := 'False'} : Bool;
         xSpare23 { ExternalWritable := 'False'} : Bool;
         xSpare24 { ExternalWritable := 'False'} : Bool;
         xSpare25 { ExternalWritable := 'False'} : Bool;
         xSpare26 { ExternalWritable := 'False'} : Bool;
         xSpare27 { ExternalWritable := 'False'} : Bool;
         xSpare28 { ExternalWritable := 'False'} : Bool;
         xSpare29 { ExternalWritable := 'False'} : Bool;
         xSpare30 { ExternalWritable := 'False'} : Bool;
         xSpare31 { ExternalWritable := 'False'} : Bool;
         xSpare { ExternalWritable := 'False'} : Array[0..15] of Bool;
         iSpare0 { ExternalWritable := 'False'} : Int;
         iSpare1 { ExternalWritable := 'False'} : Int;
         iSpare2 { ExternalWritable := 'False'} : Int;
         iSpare3 { ExternalWritable := 'False'} : Int;
         iSpare4 { ExternalWritable := 'False'} : Int;
         iSpare5 { ExternalWritable := 'False'} : Int;
         iSpare6 { ExternalWritable := 'False'} : Int;
         iSpare7 { ExternalWritable := 'False'} : Int;
         iSpare8 { ExternalWritable := 'False'} : Int;
         iSpare9 { ExternalWritable := 'False'} : Int;
         iSpare10 { ExternalWritable := 'False'} : Int;
         iSpare11 { ExternalWritable := 'False'} : Int;
         iSpare12 { ExternalWritable := 'False'} : Int;
         iSpare13 { ExternalWritable := 'False'} : Int;
         iSpare14 { ExternalWritable := 'False'} : Int;
         iSpare15 { ExternalWritable := 'False'} : Int;
         iSpare16 { ExternalWritable := 'False'} : Int;
         dZoneMode { ExternalWritable := 'False'} : DInt;   // Zone modality (1=Manual;4=Automatic;8=Manual request) {x|x|x|x|O}
         dProdModeRequest { ExternalWritable := 'False'} : DInt;   // Production modality request (1=Out of Production 3= In production) {x|x|x|x|O}
         dProdModeActual { ExternalWritable := 'False'} : DInt;   // Production modality actual (1=Out of production 3=In production 8=Out of production request 9=In production request) {x|x|x|x|O}
         dActualDistanceFromSnaproll { ExternalWritable := 'False'} : DInt;   // Actual distance from snaproll [mm/100] {x|x|x|x|O}
         dSprayCounter { ExternalWritable := 'False'} : DInt;
         dPhSprayCounter { ExternalWritable := 'False'} : DInt;
         dEvReactionTime { ExternalWritable := 'False'} : DInt;
         dCalibDeltaXPosition_cmm { ExternalWritable := 'False'} : DInt;   // Calibration.Theorical spray position X [mm/100] {mm/100|mm|0|7000|M}
         dCalibDeltaYPosition_cmm { ExternalWritable := 'False'} : DInt;   // Calibration.Theorical spray position Y [mm/100] {mm/100|mm|0|7000|M}
         dSpare9 { ExternalWritable := 'False'} : DInt;
         dSpare10 { ExternalWritable := 'False'} : DInt;
         dSpare11 { ExternalWritable := 'False'} : DInt;
         dSpare12 { ExternalWritable := 'False'} : DInt;
         dSpare13 { ExternalWritable := 'False'} : DInt;
         dSpare14 { ExternalWritable := 'False'} : DInt;
         dSpare15 { ExternalWritable := 'False'} : DInt;
         rSpare0 { ExternalWritable := 'False'} : Real;
         rSpare1 { ExternalWritable := 'False'} : Real;
         rSpare2 { ExternalWritable := 'False'} : Real;
         rSpare3 { ExternalWritable := 'False'} : Real;
         rSpare4 { ExternalWritable := 'False'} : Real;
         rSpare5 { ExternalWritable := 'False'} : Real;
         rSpare6 { ExternalWritable := 'False'} : Real;
         rSpare7 { ExternalWritable := 'False'} : Real;
         rSpare8 { ExternalWritable := 'False'} : Real;
         tManCmd { ExternalWritable := 'False'} : Struct
            xSpare0 { ExternalWritable := 'False'} : Bool;   //
            xSpare1 { ExternalWritable := 'False'} : Bool;
            xSpare2 { ExternalWritable := 'False'} : Bool;
            xSpare3 { ExternalWritable := 'False'} : Bool;
            xSpare4 { ExternalWritable := 'False'} : Bool;
            xSpare5 { ExternalWritable := 'False'} : Bool;
            xSpare6 { ExternalWritable := 'False'} : Bool;
            xSpare7 { ExternalWritable := 'False'} : Bool;
            xSpare8 { ExternalWritable := 'False'} : Bool;
            xSpare9 { ExternalWritable := 'False'} : Bool;
            xSpare10 { ExternalWritable := 'False'} : Bool;
            xSpare11 { ExternalWritable := 'False'} : Bool;
            xSpare12 { ExternalWritable := 'False'} : Bool;
            xSpare13 { ExternalWritable := 'False'} : Bool;
            xSpare14 { ExternalWritable := 'False'} : Bool;
            xSpare15 { ExternalWritable := 'False'} : Bool;
            xSpare { ExternalWritable := 'False'} : Array[0..15] of Bool;
         END_STRUCT;
      END_STRUCT;
      tHMW : Struct   // HMI Write
         xAutoModeReq : Bool;   // Automatic mode request {x|x|x|x|O}
         xManModeReq : Bool;   // Manual mode request {x|x|x|x|O}
         xUpdateDistanceFromSnapRoll : Bool;   // Update Distance From Snap Roll {x|x|x|x|M}
         xCalibrate : Bool;   // Calibrate spray position {x|x|x|x|M}
         xCleaningCycle : Bool;   // Cleaning cycle enabled {x|x|x|x|O}
         xSprayOnBreakEnabled : Bool;   // Spray during glass break {x|x|x|x|O}
         xSprayCheckEnabled : Bool;   // Spray check enabled {x|x|x|x|O}
         xResetCounter : Bool;
         xSpare8 : Bool;
         xSpare9 { ExternalWritable := 'False'} : Bool;
         xSpare10 : Bool;
         xSpare11 : Bool;
         xSpare12 : Bool;
         xSpare13 : Bool;
         xSpare14 : Bool;
         xSpare15 : Bool;   //
         xSpare16 : Bool;   //
         xSpare17 : Bool;
         xSpare18 : Bool;
         xSpare19 : Bool;
         xSpare20 : Bool;
         xSpare21 : Bool;
         xSpare22 : Bool;
         xSpare23 : Bool;
         xSpare24 : Bool;
         xSpare25 : Bool;
         xSpare26 : Bool;
         xSpare27 : Bool;
         xSpare28 : Bool;
         xSpare29 : Bool;
         xSpare30 : Bool;
         xSpare31 : Bool;
         xSpare : Array[0..15] of Bool;
         iSpare0 : Int;
         iSpare1 : Int;
         iSpare2 : Int;
         iSpare3 : Int;
         iSpare4 : Int;
         iSpare5 : Int;
         iSpare6 : Int;
         iSpare7 : Int;
         iSpare8 : Int;
         iSpare9 : Int;
         iSpare10 : Int;
         iSpare11 : Int;
         iSpare12 : Int;
         iSpare13 : Int;
         iSpare14 : Int;
         iSpare15 : Int;
         iSpare16 : Int;
         dDistanceFromSnaproll_cmm : DInt;   // Distance from snaproll [mm/100] {x|x|x|x|O}
         dSpare1 : DInt;   //
         dCleaningInterval_ms : DInt;   // Cleaning cycle interval [ms] {ms|s|3600|36000|O}
         dSpraySpace_cmm : DInt;   // Spray space [mm/100] {mm/100|mm|1|100|O}
         dSprayReactionTimeON_ms : DInt;   // Spray reaction time [ms] {ms|s|0.001|2|M}
         dSprayReactionTimeOFF_ms : DInt;   // Spray reaction time off [ms] {ms|s|0.001|2|M}
         dCalibDefectMeasXPosition_cmm : DInt;   // Calibration.Measured defect position X [mm/100] {mm/100|mm|0|7000|M}
         dCalibSprayMeasXPosition_cmm : DInt;   // Calibration.Measured spray position X [mm/100] {mm/100|mm|0|7000|M}
         dCalibDefectMeasYPosition_cmm : DInt;   // Calibration.Measured defect position Y [mm/100] {mm/100|mm|0|7000|M}
         dCalibSprayMeasYPosition_cmm : DInt;   // Calibration.Measured spray position Y [mm/100] {mm/100|mm|0|7000|M}
         dSpare10 : DInt;
         dSpare11 : DInt;
         dSpare12 : DInt;
         dSpare13 : DInt;
         dSpare14 : DInt;
         dSpare15 : DInt;
         dSpare16 : DInt;
         rSpare0 : Real;
         rSpare1 : Real;
         rSpare2 : Real;
         rSpare3 : Real;
         rSpare4 : Real;
         rSpare5 : Real;
         rSpare6 : Real;
         rSpare7 : Real;
         rSpare8 : Real;
         tManCmd : Struct
            xSpare0 : Bool;
            xSpare1 : Bool;
            xSpare2 { ExternalWritable := 'False'} : Bool;
            xSpare3 { ExternalWritable := 'False'} : Bool;
            xSpare4 { ExternalWritable := 'False'} : Bool;
            xSpare5 { ExternalWritable := 'False'} : Bool;
            xSpare6 { ExternalWritable := 'False'} : Bool;
            xSpare7 { ExternalWritable := 'False'} : Bool;
            xSpare8 { ExternalWritable := 'False'} : Bool;
            xSpare9 { ExternalWritable := 'False'} : Bool;
            xSpare10 { ExternalWritable := 'False'} : Bool;
            xSpare11 { ExternalWritable := 'False'} : Bool;
            xSpare12 { ExternalWritable := 'False'} : Bool;
            xSpare13 { ExternalWritable := 'False'} : Bool;
            xSpare14 { ExternalWritable := 'False'} : Bool;
            xSpare15 { ExternalWritable := 'False'} : Bool;
            xSpare16 : Bool;
            xSpare17 : Bool;
            xSpare18 : Bool;
            xSpare19 : Bool;
            xSpare20 : Bool;
            xSpare21 : Bool;
            xSpare22 : Bool;
            xSpare23 : Bool;
            xSpare24 : Bool;
            xSpare25 : Bool;
            xSpare26 : Bool;
            xSpare27 : Bool;
            xSpare28 : Bool;
            xSpare29 : Bool;
            xSpare30 : Bool;
            xSpare31 : Bool;
         END_STRUCT;
      END_STRUCT;
   END_STRUCT;


BEGIN
   tAlm.tE.xSpare_0 := TRUE;
   tAlm.tE.xSpare_1 := TRUE;
   tAlm.tE.xSpare_2 := TRUE;
   tAlm.tE.xSpare_3 := TRUE;
   tAlm.tE.xSpare_4 := TRUE;
   tAlm.tE.xSpare_5 := TRUE;
   tAlm.tE.xSpare_6 := TRUE;
   tAlm.tE.xSpare_7 := TRUE;
   tAlm.tE.xSpare_8 := TRUE;
   tAlm.tE.xSpare_9 := TRUE;
   tAlm.tE.xSpare_10 := FALSE;
   tAlm.tE.xSpare_11 := FALSE;
   tAlm.tE.xSpare_12 := FALSE;
   tAlm.tE.xSpare_13 := FALSE;
   tAlm.tE.xSpare_14 := FALSE;
   tAlm.tE.xSpare_15 := FALSE;
   tAlm.tE.xSpare_16 := FALSE;
   tAlm.tE.xSpare_17 := FALSE;
   tAlm.tE.xSpare_18 := FALSE;
   tAlm.tE.xSpare_19 := FALSE;
   tAlm.tE.xSpare_20 := FALSE;
   tAlm.tE.xSpare_21 := FALSE;
   tAlm.tE.xSpare_22 := FALSE;
   tAlm.tE.xSpare_23 := FALSE;
   tAlm.tE.xSpare_24 := FALSE;
   tAlm.tE.xSpare_25 := FALSE;
   tAlm.tE.xSpare_26 := FALSE;
   tAlm.tE.xSpare_27 := FALSE;
   tAlm.tE.xSpare_28 := FALSE;
   tAlm.tE.xSpare_29 := FALSE;
   tAlm.tE.xSpare_30 := FALSE;
   tAlm.tE.xSpare_31 := FALSE;
   tAlm.tS.xSpare_0 := FALSE;
   tAlm.tS.xSpare_1 := FALSE;
   tAlm.tS.xSpare_2 := FALSE;
   tAlm.tS.xSpare_3 := FALSE;
   tAlm.tS.xSpare_4 := FALSE;
   tAlm.tS.xSpare_5 := FALSE;
   tAlm.tS.xSpare_6 := FALSE;
   tAlm.tS.xSpare_7 := FALSE;
   tAlm.tS.xSpare_8 := FALSE;
   tAlm.tS.xSpare_9 := FALSE;
   tAlm.tS.xSpare_10 := FALSE;
   tAlm.tS.xSpare_11 := FALSE;
   tAlm.tS.xSpare_12 := FALSE;
   tAlm.tS.xSpare_13 := FALSE;
   tAlm.tS.xSpare_14 := FALSE;
   tAlm.tS.xSpare_15 := FALSE;
   tAlm.tS.xSpare_16 := FALSE;
   tAlm.tS.xSpare_17 := FALSE;
   tAlm.tS.xSpare_18 := FALSE;
   tAlm.tS.xSpare_19 := FALSE;
   tAlm.tS.xSpare_20 := FALSE;
   tAlm.tS.xSpare_21 := FALSE;
   tAlm.tS.xSpare_22 := FALSE;
   tAlm.tS.xSpare_23 := FALSE;
   tAlm.tS.xSpare_24 := FALSE;
   tAlm.tS.xSpare_25 := FALSE;
   tAlm.tS.xSpare_26 := FALSE;
   tAlm.tS.xSpare_27 := FALSE;
   tAlm.tS.xSpare_28 := FALSE;
   tAlm.tS.xSpare_29 := FALSE;
   tAlm.tS.xSpare_30 := FALSE;
   tAlm.tS.xSpare_31 := FALSE;
   tAlm.tF.xSpare_3 := FALSE;
   tAlm.tF.xSpare_4 := FALSE;
   tAlm.tF.xSpare_5 := FALSE;
   tAlm.tF.xSpare_6 := FALSE;
   tAlm.tF.xSpare_7 := FALSE;
   tAlm.tF.xSpare_8 := FALSE;
   tAlm.tF.xSpare_9 := FALSE;
   tAlm.tF.xSpare_10 := FALSE;
   tAlm.tF.xSpare_11 := FALSE;
   tAlm.tF.xSpare_20 := FALSE;
   tAlm.tF.xSpare_21 := FALSE;
   tAlm.tF.xSpare_22 := FALSE;
   tAlm.tF.xSpare_23 := FALSE;
   tAlm.tF.xSpare_24 := FALSE;
   tAlm.tF.xSpare_25 := FALSE;
   tAlm.tF.xSpare_26 := FALSE;
   tAlm.tF.xSpare_27 := FALSE;
   tAlm.tF.xSpare_28 := FALSE;
   tAlm.tF.xSpare_29 := FALSE;
   tAlm.tF.xSpare_30 := FALSE;
   tAlm.tF.xSpare_31 := FALSE;
   tAlm.tW.xSpare_0 := FALSE;
   tAlm.tW.xSpare_1 := FALSE;
   tAlm.tW.xSpare_2 := FALSE;
   tAlm.tW.xSpare_3 := FALSE;
   tAlm.tW.xSpare_4 := FALSE;
   tAlm.tW.xSpare_5 := FALSE;
   tAlm.tW.xSpare_6 := FALSE;
   tAlm.tW.xSpare_7 := FALSE;
   tAlm.tW.xSpare_8 := FALSE;
   tAlm.tW.xSpare_9 := FALSE;
   tAlm.tW.xSpare_10 := FALSE;
   tAlm.tW.xSpare_11 := FALSE;
   tAlm.tW.xSpare_12 := FALSE;
   tAlm.tW.xSpare_13 := FALSE;
   tAlm.tW.xSpare_14 := FALSE;
   tAlm.tW.xSpare_15 := FALSE;
   tAlm.tW.xSpare_16 := FALSE;
   tAlm.tW.xSpare_17 := FALSE;
   tAlm.tW.xSpare_18 := FALSE;
   tAlm.tW.xSpare_19 := FALSE;
   tAlm.tW.xSpare_20 := FALSE;
   tAlm.tW.xSpare_21 := FALSE;
   tAlm.tW.xSpare_22 := FALSE;
   tAlm.tW.xSpare_23 := FALSE;
   tAlm.tW.xSpare_24 := FALSE;
   tAlm.tW.xSpare_25 := FALSE;
   tAlm.tW.xSpare_26 := FALSE;
   tAlm.tW.xSpare_27 := FALSE;
   tAlm.tW.xSpare_28 := FALSE;
   tAlm.tW.xSpare_29 := FALSE;
   tAlm.tW.xSpare_30 := FALSE;
   tAlm.tW.xSpare_31 := FALSE;
   tHMR.xSpare15 := FALSE;
   tHMW.xSpare15 := FALSE;
   tHMW.xSpare16 := FALSE;

END_DATA_BLOCK

DATA_BLOCK "DB_MCC1204_HMI"
{ DB_Accessible_From_OPC_UA := 'FALSE' ;
 DB_Accessible_From_Webserver := 'FALSE' ;
 S7_Optimized_Access := 'FALSE' }
VERSION : 0.1
NON_RETAIN
   STRUCT
      tAlm : Struct   // HMI Alarms
         tE : Struct
            x0 : Bool;   // KE.Local Emergency ON
            x1 : Bool;   // SB.Emergency localization
            x2 : Bool;   // SB.Emergency localization 2
            x3 : Bool;   // SB.Emergency localization 3
            x4 : Bool;
            x5 : Bool;
            x6 : Bool;
            x7 : Bool;
            x8 : Bool;
            x9 : Bool;
            x10 : Bool;
            x11 : Bool;
            x12 : Bool;
            x13 : Bool;
            x14 : Bool;
            x15 : Bool;
            x16 : Bool;
            x17 : Bool;
            x18 : Bool;
            x19 : Bool;
            x20 : Bool;
            x21 : Bool;
            x22 : Bool;
            x23 : Bool;
            x24 : Bool;
            x25 : Bool;
            x26 : Bool;
            x27 : Bool;
            x28 : Bool;
            x29 : Bool;
            x30 : Bool;
            x31 : Bool;
         END_STRUCT;
         tS : Struct
            x0 : Bool;   // L+.Input power supply
            x1 : Bool;   // QF.Power supply 24V logic
            x2 : Bool;   // Timeout receiving consumed message
            x3 : Bool;   // Mission packet lost
            x4 : Bool;   // Synchro packet lost
            x5 : Bool;   // Meter gap outside limits
            x6 : Bool;   // Main line Meter gap outside limits
            x7 : Bool;   // Timeout receiving meter signal from main line
            x8 : Bool;   // Timeout receiving synchro value from main line
            x9 : Bool;   // Unexpected synchro pulse
            x10 : Bool;   // Unexpected synchro message
            x11 : Bool;   // Machine not synchronized
            x12 : Bool;   // SP.Missing air
            x13 : Bool;   // QF.Power supply 24V logic 2
            x14 : Bool;   // L+.Field input power supply
            x15 : Bool;   // L+.24VDC ON
            x16 : Bool;
            x17 : Bool;
            x18 : Bool;
            x19 : Bool;
            x20 : Bool;
            x21 : Bool;
            x22 : Bool;
            x23 : Bool;
            x24 : Bool;
            x25 : Bool;
            x26 : Bool;
            x27 : Bool;
            x28 : Bool;
            x29 : Bool;
            x30 : Bool;
            x31 : Bool;
         END_STRUCT;
         tF : Struct
            x0 : Bool;   // QF.Anomaly alimentation 120/230VAC
            x1 : Bool;
            x2 : Bool;
            x3 : Bool;
            x4 : Bool;
            x5 : Bool;
            x6 : Bool;
            x7 : Bool;
            x8 : Bool;
            x9 : Bool;
            x10 : Bool;
            x11 : Bool;
            x12 : Bool;
            x13 : Bool;
            x14 : Bool;
            x15 : Bool;
            x16 : Bool;
            x17 : Bool;
            x18 : Bool;
            x19 : Bool;
            x20 : Bool;
            x21 : Bool;
            x22 : Bool;
            x23 : Bool;
            x24 : Bool;
            x25 : Bool;
            x26 : Bool;
            x27 : Bool;
            x28 : Bool;
            x29 : Bool;
            x30 : Bool;
            x31 : Bool;
         END_STRUCT;
         tW : Struct
            x0 : Bool;   // A154AP1.PLCA.Timeout receiving consumed message
            x1 : Bool;   // A154AP2.PLCB.Timeout receiving consumed message
            x2 : Bool;   // A154AP1.PLCA.Mission packet lost
            x3 : Bool;   // A154AP2.PLCB.Mission packet lost
            x4 : Bool;   // A154AP1.PLCA.Syncro packet lost
            x5 : Bool;   // A154AP2.PLCB.Syncro packet lost
            x6 : Bool;
            x7 : Bool;
            x8 : Bool;
            x9 : Bool;
            x10 : Bool;
            x11 : Bool;
            x12 : Bool;
            x13 : Bool;
            x14 : Bool;
            x15 : Bool;
            x16 : Bool;
            x17 : Bool;
            x18 : Bool;
            x19 : Bool;
            x20 : Bool;
            x21 : Bool;
            x22 : Bool;
            x23 : Bool;
            x24 : Bool;
            x25 : Bool;
            x26 : Bool;
            x27 : Bool;
            x28 : Bool;
            x29 : Bool;
            x30 : Bool;
            x31 : Bool;
         END_STRUCT;
      END_STRUCT;
      tHMR { ExternalWritable := 'False'} : Struct   // HMI Read
         xSpare0 { ExternalWritable := 'False'} : Bool;
         xSpare1 { ExternalWritable := 'False'} : Bool;
         xSpare2 { ExternalWritable := 'False'} : Bool;
         xSpare3 { ExternalWritable := 'False'} : Bool;
         xSpare4 { ExternalWritable := 'False'} : Bool;
         xSpare5 { ExternalWritable := 'False'} : Bool;
         xSpare6 { ExternalWritable := 'False'} : Bool;
         xSpare7 { ExternalWritable := 'False'} : Bool;
         xSpare8 { ExternalWritable := 'False'} : Bool;
         xSpare9 { ExternalWritable := 'False'} : Bool;
         xSpare10 { ExternalWritable := 'False'} : Bool;
         xSpare11 { ExternalWritable := 'False'} : Bool;
         xSpare12 { ExternalWritable := 'False'} : Bool;
         xSpare13 { ExternalWritable := 'False'} : Bool;
         xSpare14 { ExternalWritable := 'False'} : Bool;
         xZoneAlarm { ExternalWritable := 'False'} : Bool;   // Zone alarm {X|X|X|X|O}
         xSpare16 { ExternalWritable := 'False'} : Bool;
         xSpare17 { ExternalWritable := 'False'} : Bool;
         xSpare18 { ExternalWritable := 'False'} : Bool;
         xSpare19 { ExternalWritable := 'False'} : Bool;
         xSpare20 { ExternalWritable := 'False'} : Bool;
         xSpare21 { ExternalWritable := 'False'} : Bool;
         xSpare22 { ExternalWritable := 'False'} : Bool;
         xSpare23 { ExternalWritable := 'False'} : Bool;
         xSpare24 { ExternalWritable := 'False'} : Bool;
         xSpare25 { ExternalWritable := 'False'} : Bool;
         xSpare26 { ExternalWritable := 'False'} : Bool;
         xSpare27 { ExternalWritable := 'False'} : Bool;
         xSpare28 { ExternalWritable := 'False'} : Bool;
         xSpare29 { ExternalWritable := 'False'} : Bool;
         xSpare30 { ExternalWritable := 'False'} : Bool;
         xSpare31 { ExternalWritable := 'False'} : Bool;
         xSpare { ExternalWritable := 'False'} : Array[0..15] of Bool;
         iSpare0 { ExternalWritable := 'False'} : Int;
         iSpare1 { ExternalWritable := 'False'} : Int;
         iSpare2 { ExternalWritable := 'False'} : Int;
         iSpare3 { ExternalWritable := 'False'} : Int;
         iSpare4 { ExternalWritable := 'False'} : Int;
         iSpare5 { ExternalWritable := 'False'} : Int;
         iSpare6 { ExternalWritable := 'False'} : Int;
         iSpare7 { ExternalWritable := 'False'} : Int;
         iSpare8 { ExternalWritable := 'False'} : Int;
         iSpare9 { ExternalWritable := 'False'} : Int;
         iSpare10 { ExternalWritable := 'False'} : Int;
         iSpare11 { ExternalWritable := 'False'} : Int;
         iSpare12 { ExternalWritable := 'False'} : Int;
         iSpare13 { ExternalWritable := 'False'} : Int;
         iSpare14 { ExternalWritable := 'False'} : Int;
         iSpare15 { ExternalWritable := 'False'} : Int;
         iSpare16 { ExternalWritable := 'False'} : Int;
         dSpare0 { ExternalWritable := 'False'} : DInt;
         dSpare1 { ExternalWritable := 'False'} : DInt;   // Zone status (1=CycleON 2=StopCyc 4=CycleReq 8=StopReq 1024=E-Stop) {X|X|X|X|O}
         dCabinetStatusMCC { ExternalWritable := 'False'} : DInt;   // Cabinet status MCC1201 (1=OK;2=General power alarm;3=Local power alarm) {X|X|X|X|O}
         dSpare3 { ExternalWritable := 'False'} : DInt;   //
         dSpare4 { ExternalWritable := 'False'} : DInt;   //
         dSpare5 { ExternalWritable := 'False'} : DInt;
         dSpare6 { ExternalWritable := 'False'} : DInt;
         dSpare7 { ExternalWritable := 'False'} : DInt;
         dSpare8 { ExternalWritable := 'False'} : DInt;
         dSpare9 { ExternalWritable := 'False'} : DInt;
         dSpare10 { ExternalWritable := 'False'} : DInt;
         dSpare11 { ExternalWritable := 'False'} : DInt;
         dSpare12 { ExternalWritable := 'False'} : DInt;
         dSpare13 { ExternalWritable := 'False'} : DInt;
         dSpare14 { ExternalWritable := 'False'} : DInt;
         dSpare15 { ExternalWritable := 'False'} : DInt;
         rSpare0 { ExternalWritable := 'False'} : Real;
         rSpare1 { ExternalWritable := 'False'} : Real;
         rSpare2 { ExternalWritable := 'False'} : Real;
         rSpare3 { ExternalWritable := 'False'} : Real;
         rSpare4 { ExternalWritable := 'False'} : Real;
         rSpare5 { ExternalWritable := 'False'} : Real;
         rSpare6 { ExternalWritable := 'False'} : Real;
         rSpare7 { ExternalWritable := 'False'} : Real;
         rSpare8 { ExternalWritable := 'False'} : Real;
         tManCmd { ExternalWritable := 'False'} : Struct
            xSpare0 { ExternalWritable := 'False'} : Bool;   //
            xSpare1 { ExternalWritable := 'False'} : Bool;
            xSpare2 { ExternalWritable := 'False'} : Bool;
            xSpare3 { ExternalWritable := 'False'} : Bool;
            xSpare4 { ExternalWritable := 'False'} : Bool;
            xSpare5 { ExternalWritable := 'False'} : Bool;
            xSpare6 { ExternalWritable := 'False'} : Bool;
            xSpare7 { ExternalWritable := 'False'} : Bool;
            xSpare8 { ExternalWritable := 'False'} : Bool;
            xSpare9 { ExternalWritable := 'False'} : Bool;
            xSpare10 { ExternalWritable := 'False'} : Bool;
            xSpare11 { ExternalWritable := 'False'} : Bool;
            xSpare12 { ExternalWritable := 'False'} : Bool;
            xSpare13 { ExternalWritable := 'False'} : Bool;
            xSpare14 { ExternalWritable := 'False'} : Bool;
            xSpare15 { ExternalWritable := 'False'} : Bool;
            xSpare { ExternalWritable := 'False'} : Array[0..15] of Bool;
         END_STRUCT;
      END_STRUCT;
      tHMW : Struct   // HMI Write
         xSpare0 : Bool;   //
         xSpare1 : Bool;
         xSpare2 : Bool;
         xSpare3 : Bool;
         xSpare4 : Bool;
         xSpare5 : Bool;
         xSpare6 : Bool;
         xSpare7 : Bool;
         xSpare8 : Bool;
         xSpare9 { ExternalWritable := 'False'} : Bool;
         xSpare10 : Bool;
         xSpare11 : Bool;
         xSpare12 : Bool;
         xSpare13 : Bool;
         xSpare14 : Bool;
         xFaultsReset : Bool;   // Reset faults {X|X|X|X|O}
         xGeneralReset : Bool;   // General reset {X|X|X|X|M}
         xSpare17 : Bool;
         xSpare18 : Bool;
         xSpare19 : Bool;
         xSpare20 : Bool;
         xSpare21 : Bool;
         xSpare22 : Bool;
         xSpare23 : Bool;
         xSpare24 : Bool;
         xSpare25 : Bool;
         xSpare26 : Bool;
         xSpare27 : Bool;
         xSpare28 : Bool;
         xSpare29 : Bool;
         xSpare30 : Bool;
         xSpare31 : Bool;
         xSpare : Array[0..15] of Bool;
         iSpare0 : Int;
         iSpare1 : Int;
         iSpare2 : Int;
         iSpare3 : Int;
         iSpare4 : Int;
         iSpare5 : Int;
         iSpare6 : Int;
         iSpare7 : Int;
         iSpare8 : Int;
         iSpare9 : Int;
         iSpare10 : Int;
         iSpare11 : Int;
         iSpare12 : Int;
         iSpare13 : Int;
         iSpare14 : Int;
         iSpare15 : Int;
         iSpare16 : Int;
         dSpare0 : DInt;
         dSpare1 : DInt;
         dSpare2 : DInt;   //
         dSpare3 : DInt;
         dSpare4 : DInt;
         dSpare5 : DInt;
         dSpare6 : DInt;
         dSpare7 : DInt;
         dSpare8 : DInt;
         dSpare9 : DInt;
         dSpare10 : DInt;
         dSpare11 : DInt;
         dSpare12 : DInt;
         dSpare13 : DInt;
         dSpare14 : DInt;
         dSpare15 : DInt;
         dSpare16 : DInt;
         rSpare0 : Real;
         rSpare1 : Real;
         rSpare2 : Real;
         rSpare3 : Real;
         rSpare4 : Real;
         rSpare5 : Real;
         rSpare6 : Real;
         rSpare7 : Real;
         rSpare8 : Real;
         tManCmd : Struct
            xSpare0 : Bool;   //
            xSpare1 : Bool;
            xSpare2 : Bool;
            xSpare3 : Bool;
            xSpare4 : Bool;
            xSpare5 : Bool;
            xSpare6 : Bool;
            xSpare7 : Bool;
            xSpare8 : Bool;
            xSpare9 : Bool;
            xSpare10 : Bool;
            xSpare11 : Bool;
            xSpare12 : Bool;
            xSpare13 : Bool;
            xSpare14 : Bool;
            xSpare15 : Bool;
            xSpare16 : Bool;
            xSpare17 : Bool;
            xSpare18 : Bool;
            xSpare19 : Bool;
            xSpare20 : Bool;
            xSpare21 : Bool;
            xSpare22 : Bool;
            xSpare23 : Bool;
            xSpare24 : Bool;
            xSpare25 : Bool;
            xSpare26 : Bool;
            xSpare27 : Bool;
            xSpare28 : Bool;
            xSpare29 : Bool;
            xSpare30 : Bool;
            xSpare31 : Bool;
         END_STRUCT;
      END_STRUCT;
   END_STRUCT;


BEGIN
   tAlm.tE.x0 := FALSE;
   tAlm.tE.x1 := FALSE;
   tAlm.tE.x2 := FALSE;
   tAlm.tE.x3 := FALSE;
   tAlm.tE.x4 := FALSE;
   tAlm.tE.x5 := FALSE;
   tAlm.tE.x6 := FALSE;
   tAlm.tE.x7 := FALSE;
   tAlm.tE.x8 := FALSE;
   tAlm.tE.x9 := FALSE;
   tAlm.tE.x10 := FALSE;
   tAlm.tE.x11 := FALSE;
   tAlm.tE.x12 := FALSE;
   tAlm.tE.x13 := FALSE;
   tAlm.tE.x14 := FALSE;
   tAlm.tE.x15 := FALSE;
   tAlm.tE.x16 := FALSE;
   tAlm.tE.x17 := FALSE;
   tAlm.tE.x18 := FALSE;
   tAlm.tE.x19 := FALSE;
   tAlm.tE.x20 := FALSE;
   tAlm.tE.x21 := FALSE;
   tAlm.tE.x22 := FALSE;
   tAlm.tE.x23 := FALSE;
   tAlm.tE.x24 := FALSE;
   tAlm.tE.x25 := FALSE;
   tAlm.tE.x26 := FALSE;
   tAlm.tE.x27 := FALSE;
   tAlm.tE.x28 := FALSE;
   tAlm.tE.x29 := FALSE;
   tAlm.tE.x30 := FALSE;
   tAlm.tE.x31 := FALSE;
   tAlm.tS.x0 := FALSE;
   tAlm.tS.x1 := FALSE;
   tAlm.tS.x2 := FALSE;
   tAlm.tS.x3 := FALSE;
   tAlm.tS.x4 := FALSE;
   tAlm.tS.x5 := FALSE;
   tAlm.tS.x6 := FALSE;
   tAlm.tS.x7 := FALSE;
   tAlm.tS.x8 := FALSE;
   tAlm.tS.x9 := FALSE;
   tAlm.tS.x10 := FALSE;
   tAlm.tS.x11 := FALSE;
   tAlm.tS.x12 := FALSE;
   tAlm.tS.x13 := FALSE;
   tAlm.tS.x14 := FALSE;
   tAlm.tS.x15 := FALSE;
   tAlm.tS.x16 := FALSE;
   tAlm.tS.x17 := FALSE;
   tAlm.tS.x18 := FALSE;
   tAlm.tS.x19 := FALSE;
   tAlm.tS.x20 := FALSE;
   tAlm.tS.x21 := FALSE;
   tAlm.tS.x22 := FALSE;
   tAlm.tS.x23 := FALSE;
   tAlm.tS.x24 := FALSE;
   tAlm.tS.x25 := FALSE;
   tAlm.tS.x26 := FALSE;
   tAlm.tS.x27 := FALSE;
   tAlm.tS.x28 := FALSE;
   tAlm.tS.x29 := FALSE;
   tAlm.tS.x30 := FALSE;
   tAlm.tS.x31 := FALSE;
   tAlm.tF.x0 := FALSE;
   tAlm.tF.x1 := FALSE;
   tAlm.tF.x2 := FALSE;
   tAlm.tF.x3 := FALSE;
   tAlm.tF.x4 := FALSE;
   tAlm.tF.x5 := FALSE;
   tAlm.tF.x6 := FALSE;
   tAlm.tF.x7 := FALSE;
   tAlm.tF.x8 := FALSE;
   tAlm.tF.x9 := FALSE;
   tAlm.tF.x10 := FALSE;
   tAlm.tF.x11 := FALSE;
   tAlm.tF.x12 := FALSE;
   tAlm.tF.x13 := FALSE;
   tAlm.tF.x14 := FALSE;
   tAlm.tF.x15 := FALSE;
   tAlm.tF.x16 := FALSE;
   tAlm.tF.x17 := FALSE;
   tAlm.tF.x18 := FALSE;
   tAlm.tF.x19 := FALSE;
   tAlm.tF.x20 := FALSE;
   tAlm.tF.x21 := FALSE;
   tAlm.tF.x22 := FALSE;
   tAlm.tF.x23 := FALSE;
   tAlm.tF.x24 := FALSE;
   tAlm.tF.x25 := FALSE;
   tAlm.tF.x26 := FALSE;
   tAlm.tF.x27 := FALSE;
   tAlm.tF.x28 := FALSE;
   tAlm.tF.x29 := FALSE;
   tAlm.tF.x30 := FALSE;
   tAlm.tF.x31 := FALSE;
   tAlm.tW.x0 := FALSE;
   tAlm.tW.x1 := FALSE;
   tAlm.tW.x2 := FALSE;
   tAlm.tW.x3 := FALSE;
   tAlm.tW.x4 := FALSE;
   tAlm.tW.x5 := FALSE;
   tAlm.tW.x6 := FALSE;
   tAlm.tW.x7 := FALSE;
   tAlm.tW.x8 := FALSE;
   tAlm.tW.x9 := FALSE;
   tAlm.tW.x10 := FALSE;
   tAlm.tW.x11 := FALSE;
   tAlm.tW.x12 := FALSE;
   tAlm.tW.x13 := FALSE;
   tAlm.tW.x14 := FALSE;
   tAlm.tW.x15 := FALSE;
   tAlm.tW.x16 := FALSE;
   tAlm.tW.x17 := FALSE;
   tAlm.tW.x18 := FALSE;
   tAlm.tW.x19 := FALSE;
   tAlm.tW.x20 := FALSE;
   tAlm.tW.x21 := FALSE;
   tAlm.tW.x22 := FALSE;
   tAlm.tW.x23 := FALSE;
   tAlm.tW.x24 := FALSE;
   tAlm.tW.x25 := FALSE;
   tAlm.tW.x26 := FALSE;
   tAlm.tW.x27 := FALSE;
   tAlm.tW.x28 := FALSE;
   tAlm.tW.x29 := FALSE;
   tAlm.tW.x30 := FALSE;
   tAlm.tW.x31 := FALSE;
   tHMR.xZoneAlarm := FALSE;
   tHMR.dSpare1 := 1024;
   tHMR.dCabinetStatusMCC := 1;
   tHMW.xSpare5 := FALSE;
   tHMW.xSpare6 := FALSE;
   tHMW.xSpare7 := FALSE;
   tHMW.xFaultsReset := FALSE;
   tHMW.xGeneralReset := FALSE;

END_DATA_BLOCK

